{attribute 'GeneratedUsingTerminal: EL5151-0080-0016'}
{attribute addProperty BoxType "EL5151-0080-0016"}
{attribute addProperty Id "Latch_C_validAT %I*BOOL1Latch_extern_validAT %I*BOOL1Set_counter_doneAT %I*BOOL1Extrapolation_stallAT %I*BOOL1Status_of_input_AAT %I*BOOL1Status_of_input_BAT %I*BOOL1Status_of_input_CAT %I*BOOL1Status_of_extern_latchAT %I*BOOL1Sync_ErrorAT %I*BOOL1TxPDO_ToggleAT %I*BOOL1Counter_valueAT %I*UINT2Latch_valueAT %I*UINT2"}
{attribute addProperty CRC "4047062379"}
{attribute addProperty Size "14"}
TYPE ENC_Inputs_F139456B :
STRUCT
	{attribute addProperty Name "Latch_C_valid"}
	Latch_C_valid AT %I* : BOOL;
	{attribute addProperty Name "Latch_extern_valid"}
	Latch_extern_valid AT %I* : BOOL;
	{attribute addProperty Name "Set_counter_done"}
	Set_counter_done AT %I* : BOOL;
	{attribute addProperty Name "Extrapolation_stall"}
	Extrapolation_stall AT %I* : BOOL;
	{attribute addProperty Name "Status_of_input_A"}
	Status_of_input_A AT %I* : BOOL;
	{attribute addProperty Name "Status_of_input_B"}
	Status_of_input_B AT %I* : BOOL;
	{attribute addProperty Name "Status_of_input_C"}
	Status_of_input_C AT %I* : BOOL;
	{attribute addProperty Name "Status_of_extern_latch"}
	Status_of_extern_latch AT %I* : BOOL;
	{attribute addProperty Name "Sync_Error"}
	Sync_Error AT %I* : BOOL;
	{attribute addProperty Name "TxPDO_Toggle"}
	TxPDO_Toggle AT %I* : BOOL;
	{attribute addProperty Name "Counter_value"}
	Counter_value AT %I* : UINT;
	{attribute addProperty Name "Latch_value"}
	Latch_value AT %I* : UINT;
END_STRUCT
END_TYPE

(* stored: Version 1.2.0.0, ProductVersion 3.1.4024.9
   DUT ENC_Inputs_F139456B: Id {734153bb-9767-47b7-bc88-359f973e7f34} *)
